(* IEC 61131-3 sources: github/ST定义, 5 files *)

(* ---- 座台定义.st ---- *)
TYPE E_NozzleState :
(
    (* 状态机枚举 *)
	eState_Idle,				// 空闲状态
	eState_Init,				// 初始化
	eState_NozzleIning,			// 座台进中(2段)
	eState_NozzleIned,			// 座台进完成
	eState_NozzleOuting,		// 座台退中(2段)
	eState_NozzleOuted,			// 座台退完成
	eState_Error				// 错误状态

);
END_TYPE

TYPE ST_NozzleSeg :
STRUCT

	(* 单段工艺参数 *)
	uiPres: UINT;		// 设定压力
	uiSpd: UINT;		// 设定速度
	udiPos: UDINT;		// 设定位置
	uiTime: UINT;		// 设定时间
	uiPresGrad: UINT;	// 设定压力斜率
	uiSpdGrad: UINT;	// 设定速度斜率

END_STRUCT
END_TYPE

TYPE ST_NozzlePara :
STRUCT

	(* 座台进工艺参数 21*)
	uiNozzleInSegCnt: UINT;							// 座台进段数选择
	uiNozzleInMode: UINT;							// 座台进方式选择 0:时间  1:行程  2:位置
	uiNozzleInLimitTime: UINT;						// 座台进限制时间
	aNozzleInSeg: ARRAY[1..2] OF ST_NozzleSeg;		// 座台进多段设定参数

	uiNozzleInPresStartGrad: UINT;				// 压力启动斜率
	uiNozzleInPresStopGrad: UINT;				// 压力停止斜率
	uiNozzleInSpdStartGrad: UINT;				// 速度启动斜率
	uiNozzleInSpdStopGrad: UINT;				// 速度停止斜率

	(* 座台退工艺参数 21*)
	uiNozzleOutSegCnt: UINT;							// 座台退段数选择
	uiNozzleOutMode: UINT;							// 座台退方式选择 0:时间  1:行程  2:位置
	uiNozzleOutLimitTime: UINT;						// 座台退限制时间
	aNozzleOutSeg: ARRAY[1..2] OF ST_NozzleSeg;		// 座台退多段设定参数

	uiNozzleOutPresStartGrad: UINT;				// 压力启动斜率
	uiNozzleOutPresStopGrad: UINT;				// 压力停止斜率
	uiNozzleOutSpdStartGrad: UINT;				// 速度启动斜率
	uiNozzleOutSpdStopGrad: UINT;				// 速度停止斜率

	(* 座台调试模式参数（调模状态下使用） *)
	stNozzleInDbgSeg: ST_NozzleSeg;				// 座台进调试段参数
	stNozzleOutDbgSeg: ST_NozzleSeg;			// 座台退调试段参数

END_STRUCT
END_TYPE

VAR_IN_OUT
	stNozzleAxis: ST_AxisRefHyd;
END_VAR
VAR_INPUT

    (* 控制命令 *)
	bStart: BOOL;				// 启动
	bStop: BOOL;				// 停止(有减速停)
	bEStop: BOOL;				// 急停(立即停止，无减速停)
	bReset: BOOL;				// 复位

    (* 模式选择 *)
	uiNozzleMode: UINT;		// 0:无模式 1:座台进模式 2:座台退模式 3:座台进(调试模式) 4:座台退(调试模式)

	(* 上位机设定参数输入 *)
	stNozzlePara: ST_NozzlePara;

	(* 数字信号输入 *)
	bNozzleInStop: BOOL;			// 座台进停止
	bNozzleOutStop: BOOL;			// 座台退停止

	(* 模拟信号输入 *)
	udiNozzleElecRulerVal: UDINT;			// 座台电子尺值

END_VAR
VAR_OUTPUT

	(* 状态输出 *)
	bBusy: BOOL;		// 忙状态
	bDone: BOOL;		// 完成状态
	bAlarm: BOOL;		// 报警状态

    (* 报警信息 *)
	dwAlarmID: DWORD;		// 报警代码（按位标识，可同时报告多个报警）
							(*	Bit0(1):   座台进超时
								Bit1(2):   座台退超时
								Bit2(4):   位置超限
								Bit3(8):   传感器异常
								...其他位预留
							*)

    (* 动作提示 *)
	uiActHint: UINT;		// 当前动作状态
							(*	0:无动作	1:报警状态	  2:座台进完成  3:座台退完成
								10: 		11:座台进1段  12:座台进2段	13:
								20:			21:座台退1段  22:座台退2段  23:
							*)
	uiActTime: UINT;		// 当前动作运行时间

	(* 动作状态输出 *)
	bNozzleIned: BOOL;		// 座台进完成
	bNozzleOuted: BOOL;		// 座台退完成

    (* 控制命令输出 *)
	uiPresCmd: UINT;		// 压力命令输出
	uiSpdCmd: UINT;			// 速度命令输出
	udiPosCmd: UDINT;		// 位置命令输出

END_VAR

(* ---- 储料定义.st ---- *)
TYPE E_MeterState :
(
    (* 状态机枚举 *)
	eState_Idle,				// 空闲状态
	eState_Init,				// 初始化
	eState_Metering,			// 储料中(8段)
	eState_Metered,				// 储料完成
	eState_Error				// 错误状态

);
END_TYPE

TYPE ST_MeterSeg :
STRUCT

	(* 单段工艺参数 *)
	uiSPres: UINT;		// 设定压力
	uiBackPres: UINT;	// 设定背压
	uiSpd: UINT;		// 设定速度
	udiPos: UDINT;		// 设定位置
	uiPresGrad: UINT;	// 设定压力斜率
	uiSpdGrad: UINT;	// 设定速度斜率

END_STRUCT
END_TYPE

TYPE ST_MeterPara :
STRUCT

	(* 储料工艺参数 71*)
	uiMeterSegCnt: UINT;						// 储料段数选择
	uiMeterMode: UINT;							// 储料退方式选择 0:电子尺  1:行程
	uiMeterLimitTime: UINT;						// 储料限制时间
	aMeterSeg: ARRAY[1..8] OF ST_MeterSeg;		// 储料多段设定参数

	uiMeterPresStartGrad: UINT;			// 压力启动斜率
	uiMeterPresStopGrad: UINT;			// 压力停止斜率
	uiMeterSpdStartGrad: UINT;			// 速度启动斜率
	uiMeterSpdStopGrad: UINT;			// 速度停止斜率

END_STRUCT
END_TYPE

FUNCTION_BLOCK FB_Meter
VAR_IN_OUT
	stMeterAxis: ST_AxisRefHyd;
END_VAR
VAR_INPUT

    (* 控制命令 *)
	bStart: BOOL;				// 启动
	bStop: BOOL;				// 停止(有减速停)
	bEStop: BOOL;				// 急停(立即停止，无减速停)
	bReset: BOOL;				// 复位

    (* 模式选择 *)
// 	uiMeterMode: UINT;		// 0:无模式 1: 2: 3:

	(* 上位机设定参数输入 *)
	stMeterPara: ST_MeterPara;

	(* 数字信号输入 *)
	bMeterStop: BOOL;			// 储料停止

	(* 模拟信号输入 *)
	udiInjElecRulerVal: UDINT;			// 射胶电子尺值

END_VAR
VAR_OUTPUT

	(* 状态输出 *)
	bBusy: BOOL;		// 忙状态
	bDone: BOOL;		// 完成状态
	bAlarm: BOOL;		// 报警状态
    (* 报警信息 *)
	dwAlarmID: DWORD;		// 报警代码（按位标识，可同时报告多个报警）
							(*	Bit0(1):   储料超时
								Bit1(2):   位置超限
								...其他位预留
							*)

    (* 动作提示 *)
	uiActHint: UINT;		// 当前动作状态
							(*	0:无动作  1:报警状态  2:储料完成    3:
								10: 	  11:储料1段  12:储料2段	13: 储料3段  14:储料4段    15:储料5段  16: 储料6段  17:储料7段   18:储料8段
							*)
	uiActTime: UINT;		// 当前动作运行时间

	(* 动作状态输出 *)
	bMetered: BOOL;				//储料完成

    (* 控制命令输出 *)
	uiPresCmd: UINT;		// 压力命令输出
	uiBackPresCmd: UINT;	// 背压命令输出
	uiSpdCmd: UINT;			// 速度命令输出
	udiPosCmd: UDINT;		// 位置命令输出

END_VAR

(* ---- 开合模定义.st ---- *)
(*
 * 文件: 开合模定义.st
 * 版本: V1.1
 *
 * 版本历史:
 * V1.0  2026-03-27  初始版本
 * V1.1  2026-04-02  新增调试模式支持(stOpenDebug/stCloseDebug)
 *
 * 说明: 开合模机构控制的功能块和数据结构定义
 *)

TYPE E_AxisState :
(
	Idle,				// 空闲状态
	Running,				// 运行状态
	Stop					// 停止状态
);
END_TYPE

TYPE E_ClampState :
(
	(* 状态机枚举 *)
	eState_Idle,				// 空闲状态
	eState_Init,				// 初始化
	eState_OpenUnload,			// 开模卸荷
	eState_Opening,				// 开模中(5段)
	eState_Opened,				// 开模完成
	eState_Closing,				// 合模中(3段)
	eState_Closed,				// 合模完成
	eState_CloseLowPress,		// 合模低压
	eState_CloseHighPress,		// 合模高压
	eState_Error				// 错误状态
);
END_TYPE

TYPE ST_PumpRequest :
STRUCT
	bRequest: BOOL;			// 泵请求
	rFlowSet: LREAL;		// 流量设定
	rPressureSet: LREAL;	// 压力设定
END_STRUCT
END_TYPE

TYPE ST_AxisRefHyd :
STRUCT
	(* 静态参数 *)
	bActive: BOOL;					// 轴是否激活
	eAxisState: E_AxisState;		// 轴状态
	nAxisID: INT;					// 轴ID号
	rMaxCylinderStroke: LREAL;		// 最大油缸行程
	rMaxVelocity: LREAL;			// 最大速度
	rMaxPressure: LREAL;			// 最大压力

	(* 运行设定值 *)
	rSetPosition: LREAL;				// 目标位置
	rSetVelocity: LREAL;			// 目标速度
	rSetPressure: LREAL;			// 目标压力

	(* 运行实际值 *)
	rActualPosition: LREAL;			// 实际位置
	rActualVelocity: LREAL;			// 实际速度
	rActualPressure: LREAL;			// 实际压力

	(* 泵请求 *)
	stPumpRequest: ST_PumpRequest;	// 向泵发送的请求

	(* 故障信息 *)
	nFaultCode: INT;					// 故障码
END_STRUCT
END_TYPE

TYPE ST_ClampSeg :
STRUCT

	(* 单段工艺参数 *)
	uiPres: UINT;		// 设定压力
	uiSpd: UINT;		// 设定速度
	udiPos: UDINT;		// 设定位置
	uiTime: UINT;		// 设定时间
	uiPresGrad: UINT;	// 设定压力斜率
	uiSpdGrad: UINT;	// 设定速度斜率

END_STRUCT
END_TYPE

TYPE ST_ClampPara :
STRUCT

	(* 开模工艺参数 *)
	uiOpenSegCnt: UINT;							// 开模段数选择 (1-5段)
	uiOpenMode: UINT;							// 开模方式选择 0:电子尺  1:行程
	uiOpenLimitTime: UINT;						// 开模限制时间
	stOpenUnloadPres: ST_ClampSeg;				// 开模卸荷设定参数
	aOpenSeg: ARRAY[1..5] OF ST_ClampSeg;		// 开模多段设定参数

	uiOpenPresStartGrad: UINT;					// 开模压力启动斜率
	uiOpenPresStopGrad: UINT;					// 开模压力停止斜率
	uiOpenSpdStartGrad: UINT;					// 开模速度启动斜率
	uiOpenSpdStopGrad: UINT;					// 开模速度停止斜率

	(* 合模工艺参数 *)
	uiCloseSegCnt: UINT;							// 合模段数选择 (1-3段)
	uiCloseMode: UINT;							// 合模方式选择 0:电子尺  1:行程
	uiCloseLimitTime: UINT;						// 合模限制时间
	uiCloseLowPresLimitTime: UINT;					// 合模低压保护时间
	uiCloseEndMode: UINT;							// 合模终止方式选择 0:时间 1:行程 2:压力
	uiCloseEndHighPres: UINT;						// 合模高压压力
	aCloseSeg: ARRAY[1..3] OF ST_ClampSeg;		// 合模多段设定参数
	stCloseLowPres: ST_ClampSeg;					// 合模低压设定参数
	stCloseHighPres: ST_ClampSeg;					// 合模高压设定参数

	uiClosePresStartGrad: UINT;					// 合模压力启动斜率
	uiClosePresStopGrad: UINT;					// 合模压力停止斜率
	uiCloseSpdStartGrad: UINT;					// 合模速度启动斜率
	uiCloseSpdStopGrad: UINT;					// 合模速度停止斜率

	(* 调试模式参数（调模状态下使用） *)
	stOpenDebug: ST_ClampSeg;					// 开模调试参数
	stCloseDebug: ST_ClampSeg;					// 合模调试参数

	(* 中子控制参数 *)
	aCoreFn: ARRAY[1..8] OF UINT;				// 中子功能 0:不使用 1:使用
	aCoreInMode: ARRAY[1..8] OF UINT;			// 中子进开始方式 0:行程 1:位置
	aCoreInStroke: ARRAY[1..8] OF UINT;		// 中子进开始行程
	aCoreInPos: ARRAY[1..8] OF UDINT;			// 中子进开始位置
	aCoreOutMode: ARRAY[1..8] OF UINT;			// 中子退开始方式 0:行程 1:位置
	aCoreOutStroke: ARRAY[1..8] OF UINT;		// 中子退开始行程
	aCoreOutPos: ARRAY[1..8] OF UDINT;			// 中子退开始位置

END_STRUCT
END_TYPE

FUNCTION_BLOCK FB_Clamp
VAR_IN_OUT
	ClampAxis: ST_AxisRefHyd;
END_VAR
VAR_INPUT

	(* 控制命令 *)
	bStart: BOOL;				// 启动
	bStop: BOOL;				// 停止(有减速停)
	bEStop: BOOL;				// 急停(立即停止，无减速停)
	bReset: BOOL;				// 复位

	(* 模式选择 *)
	uiClampMode: UINT;			// 0:无模式 1:开模模式 2:合模模式 3:开模(调试模式) 4:合模(调试模式)

	(* 上位机设定参数输入 *)
	stClampPara: ST_ClampPara;

	(* 数字信号输入 *)
	bOpenStop: BOOL;				// 开模停止
	bCloseLowPres: BOOL;			// 合模低压
	bCloseHighPres: BOOL;			// 合模高压
	bCloseStop: BOOL;				// 合模停止

	(* 模拟信号输入 *)
	udiClampElecRulerVal: UDINT;			// 锁模电子尺值
	uiClampPresElecRulerVal: UINT;			// 锁模压力值

END_VAR
VAR_OUTPUT

	(* 状态输出 *)
	bBusy: BOOL;		// 忙状态
	bDone: BOOL;		// 完成状态
	bAlarm: BOOL;		// 报警状态

	(* 报警信息 *)
	dwAlarmID: DWORD;		// 报警代码（按位标识，可同时报告多个报警）
							(*	Bit0(1):   低压保护超时
								Bit1(2):   开模超时
								Bit2(4):   合模超时
								Bit3(8):   位置超限
								Bit4(16):  传感器异常
								...其他位预留
							*)

	(* 动作提示 *)
	uiActHint: UINT;		// 当前动作状态
							(*	0:无动作	1:报警状态	2:开模完成  3:合模完成  4:中子执行
								10:开模卸荷	11:开模1段  12:开模2段	13:开模3段  14:开模4段  15:开模5段
								21:合模1段	22:合模2段  23:合模3段
								30:合模低压	31:合模高压
								40:开模调试	41:合模调试
							*)
	uiActTime: UINT;		// 当前动作运行时间
	bMoldOpened: BOOL;		// 开模完成
	bMoldClosed: BOOL;		// 合模完成
	aCoreAllow: ARRAY[1..8] OF BOOL;		// 中子允许信号（1..8组）

	(* 输出命令 *)
	uiPresCmd: UINT;		// 压力命令输出
	uiSpdCmd: UINT;		// 速度命令输出
	udiPosCmd: UDINT;		// 位置命令输出

END_VAR

(* ---- 液压伺服.st ---- *)
TYPE ST_AxisRefHyd :
STRUCT
	// ================================
	// AXIS_REF 轴索引结构体【完整版】
	// 包含：轴所有状态、位置、速度、扭矩、限位、报警、参数
	// ================================

    // ========== 1. 轴基础信息 ==========
    AxisNo           : INT;          // 轴编号 (0,1,2,3...)
    AxisName         : STRING[32];   // 轴名称
    Valid            : BOOL;         // 轴结构体有效
    AxisRefId        : UINT;         // 内部轴ID

    // ========== 2. 轴使能与状态 ==========
    Enabled          : BOOL;         // 轴已使能
    PowerOn          : BOOL;         // 伺服已上电
    Faulted          : BOOL;         // 轴故障
    Ready            : BOOL;         // 轴准备就绪
    Stopped          : BOOL;         // 轴已停止
    Moving           : BOOL;         // 轴正在运动
    Homing           : BOOL;         // 正在回零
    HomingDone       : BOOL;         // 回零完成
    InPosition       : BOOL;         // 已到达目标位置

    // ========== 3. 控制模式 ==========
    ControlMode      : INT;          // 当前控制模式
    // 0=未激活 1=位置 2=速度 3=扭矩 4=回零
    HomingMode       : INT;          // 回零模式

    // ========== 4. 位置数据 ==========
    ActualPosition   : LREAL;        // 实际位置（实时）
    CommandPosition  : LREAL;        // 指令位置
    HomePosition     : LREAL;        // 原点位置
    TargetPosition   : LREAL;        // 目标位置

    // ========== 5. 速度数据 ==========
    ActualVelocity   : LREAL;        // 实际速度
    CommandVelocity  : LREAL;        // 指令速度
    MaxVelocity      : LREAL;        // 轴最大速度

    // ========== 6. 加速度数据 ==========
    Acceleration     : LREAL;        // 当前加速度
    Deceleration     : LREAL;        // 当前减速度
    MaxAcceleration  : LREAL;        // 最大加速度
    MaxDeceleration  : LREAL;        // 最大减速度
    Jerk             : LREAL;        // 跃度
    MaxJerk          : LREAL;        // 最大跃度

    // ========== 7. 扭矩/力矩数据 ==========
    ActualTorque     : LREAL;        // 实际扭矩
    MaxTorque        : LREAL;        // 最大扭矩
    TorqueLimit      : LREAL;        // 扭矩限制

    // ========== 8. 限位信号 ==========
    PositiveLimit    : BOOL;         // 正限位触发
    NegativeLimit    : BOOL;         // 负限位触发
    SoftPlusLimit    : BOOL;         // 软正限位
    SoftNegLimit     : BOOL;         // 软负限位

    // ========== 9. 错误与报警 ==========
    Error            : BOOL;         // 轴错误
    ErrorId          : DWORD;        // 错误代码
    DriveAlarm       : BOOL;         // 驱动器报警
    DriveErrorId     : DWORD;        // 驱动器错误码
    ErrorStop        : BOOL;         // 错误停止

    // ========== 10. 状态字 ==========
    AxisStatus       : DWORD;        // 轴状态字
    DriveStatus      : DWORD;        // 驱动器状态字
    StatusBits       : ARRAY[0..15] OF BOOL; // 状态位

	(* 根据实际需求可以增加变量	*)

    // 1. 几何尺寸
    Bore_Dia        : LREAL;  // 缸径 mm
    Rod_Dia         : LREAL;  // 杆径 mm
    Stroke          : LREAL;  // 总行程 mm
    Min_Len         : LREAL;  // 最小安装距
    Max_Len         : LREAL;  // 最大安装距

    // 2. 面积容积
    Area_Piston     : LREAL;  // mm²
    Area_Rod        : LREAL;  // mm²
    Area_Annular    : LREAL;  // mm²
    Vol_Per_MM      : LREAL;  // mL/mm

    // 3. 压力推力
    Press_Rated     : LREAL;  // MPa
    Press_Max       : LREAL;  // MPa
    Force_Extend    : LREAL;  // N
    Force_Retract   : LREAL;  // N
    Effi            : LREAL;  // 效率

    // 4. 速度流量
    Vel_Ext_Max     : LREAL;  // mm/s
    Vel_Ret_Max     : LREAL;  // mm/s
    Flow_Ext        : LREAL;  // L/min
    Flow_Ret        : LREAL;  // L/min

    // 5. 位置限位
    Soft_Limit_F    : LREAL;  // 正向软限位
    Soft_Limit_B    : LREAL;  // 反向软限位
    Home_Pos        : LREAL;  // 原点位置
    Pos_Tolerance   : LREAL;  // 定位允差

    // 6. 负载摩擦
    Friction        : LREAL;
    Max_Axial_Load  : LREAL;
    Max_Rad_Load    : LREAL;

END_STRUCT
END_TYPE

FUNCTION_BLOCK FB_AxisHyd
VAR_IN_OUT
	stAxisHyd: ST_AxisRefHyd;
END_VAR
VAR_INPUT

    (* 控制命令 *)
	bStart: BOOL;		// 启动
	bStop: BOOL;		// 停止(有减速停)
	bEStop: BOOL;		// 急停(立即停止，无减速停)
	bReset: BOOL;		// 复位
	bDir: BOOL;			// 方向

    (* 模式选择 *)
	uiMode: UINT;		// 0:无模式 1:位置模式 2:速度模式 3:扭矩模式

    (* 参数设定 *)
	uiCmdPres  : UINT; 	// 压力目标
    uiSpd      : UINT; 	// 速度目标
    udiPos     : UDINT; // 位置目标
    uiForce    : UINT; 	// 力目标，可选(锁模,射胶时使用）

    uiAcc	: UINT;     // 加速度
    uiDec	: UINT;     // 减速度
	uiJerk	: UINT;     // 加加速

END_VAR
VAR_OUTPUT

	(* 状态输出 *)
	bBusy: BOOL;		// 忙状态
	bDone: BOOL;		// 完成状态
	bAlarm: BOOL;		// 报警状态

    (* 报警信息 *)
	dwAlarmID: DWORD;		// 报警代码
							(*	0:无
							*)

END_VAR
VAR
	// 状态机状态
	State: INT;
	// 内部状态
	StartOld: BOOL;
	StopOld: BOOL;
	EStopOld: BOOL;
	ResetOld: BOOL;
	// 位置/速度模拟
	SimPosition: LREAL;
	SimVelocity: LREAL;
	SimTorque: LREAL;
END_VAR

TYPE EN_AxisState =
(
	AXIS_IDLE		:= 0,	// 空闲
	AXIS_STARTING	:= 1,	// 启动中
	AXIS_RUNNING	:= 2,	// 运行中
	AXIS_STOPPING	:= 3,	// 停止中
	AXIS_STOPPED	:= 4,	// 已停止
	AXIS_ESTOPPING	:= 5,	// 急停中
	AXIS_ERROR		:= 6,	// 错误状态
	AXIS_RESETTING	:= 7	// 复位中
);
END_TYPE

(*
===================================================================
FB_AxisHyd - 液压伺服轴功能块【简化版】
===================================================================
功能：提供液压伺服轴的基本控制接口，用于PLC编程验证
备注：实际驱动器通信部分待后续实现

使用方式：
1. 配置 stAxisHyd 中的轴参数（行程、限位等）
2. 设置 uiMode 选择控制模式
3. 设置目标值（uiCmdPres, uiSpd, udiPos, uiForce）
4. 置位 bStart 启动轴运动
5. 监控 bBusy/bDone/bAlarm 状态

模式说明：
- uiMode=1: 位置模式 - 运动到 udiPos 指定位置
- uiMode=2: 速度模式 - 以 uiSpd 指定速度运动
- uiMode=3: 扭矩模式 - 以 uiForce 指定力运动
===================================================================
*)
FB_AxisHyd();

// 状态机
CASE State OF
	// ==================== 空闲状态 ====================
	AXIS_IDLE:
		bBusy		:= FALSE;
		bDone		:= FALSE;
		stAxisHyd.Moving	:= FALSE;
		stAxisHyd.Stopped	:= TRUE;

		// 检测启动命令
		IF bStart AND NOT StartOld THEN
			// 检查急停和报警
			IF stAxisHyd.DriveAlarm THEN
				dwAlarmID	:= 16#0001;	// 驱动器报警
				bAlarm		:= TRUE;
				State		:= AXIS_ERROR;
			ELSIF stAxisHyd.PositiveLimit AND bDir THEN
				dwAlarmID	:= 16#0002;	// 正限位
				bAlarm		:= TRUE;
				State		:= AXIS_ERROR;
			ELSIF stAxisHyd.NegativeLimit AND NOT bDir THEN
				dwAlarmID	:= 16#0003;	// 负限位
				bAlarm		:= TRUE;
				State		:= AXIS_ERROR;
			ELSE
				// 进入启动
				State		:= AXIS_STARTING;
			END_IF
		END_IF

	// ==================== 启动中 ====================
	AXIS_STARTING:
		bBusy		:= TRUE;
		stAxisHyd.Moving	:= TRUE;
		stAxisHyd.Stopped	:= FALSE;

		// 初始化模拟位置
		SimPosition	:= stAxisHyd.ActualPosition;
		SimVelocity	:= 0.0;
		SimTorque	:= 0.0;

		// 模式选择
		CASE uiMode OF
			1: // 位置模式
				stAxisHyd.TargetPosition	:= LREAL(udiPos) / 1000.0; // 单位转换
				stAxisHyd.CommandVelocity	:= LREAL(uiSpd) / 1000.0;
				stAxisHyd.CommandPosition	:= stAxisHyd.TargetPosition;

			2: // 速度模式
				SimVelocity	:= LREAL(uiSpd) / 1000.0;

			3: // 扭矩模式
				SimTorque	:= LREAL(uiForce) / 1000.0;

			ELSE
				dwAlarmID	:= 16#0010;	// 无效模式
				bAlarm		:= TRUE;
				State		:= AXIS_ERROR;
		END_CASE

		State	:= AXIS_RUNNING;

	// ==================== 运行中 ====================
	AXIS_RUNNING:
		bBusy		:= TRUE;
		stAxisHyd.Moving	:= TRUE;
		stAxisHyd.Stopped	:= FALSE;
		stAxisHyd.InPosition	:= FALSE;

		// 急停检测
		IF bEStop AND NOT EStopOld THEN
			State	:= AXIS_ESTOPPING;
		// 停止命令
		ELSIF bStop AND NOT StopOld THEN
			State	:= AXIS_STOPPING;
		// 位置模式到位检测
		ELSIF uiMode = 1 THEN
			SimPosition	:= SimPosition + SimVelocity * 0.05; // 模拟位置变化
			stAxisHyd.ActualPosition	:= SimPosition;

			// 到位判断
			IF ABS(SimPosition - stAxisHyd.TargetPosition) <= stAxisHyd.Pos_Tolerance THEN
				State	:= AXIS_STOPPED;
			END_IF
		// 速度/扭矩模式需要外部停止
		ELSE
			// 模拟运动
			IF bDir THEN
				SimPosition	:= SimPosition + SimVelocity * 0.05;
			ELSE
				SimPosition	:= SimPosition - SimVelocity * 0.05;
			END_IF
			stAxisHyd.ActualPosition	:= SimPosition;
		END_IF

	// ==================== 停止中 ====================
	AXIS_STOPPING:
		bBusy		:= TRUE;
		SimVelocity	:= SimVelocity * 0.8; // 减速

		IF ABS(SimVelocity) < 0.001 THEN
			SimVelocity	:= 0.0;
			stAxisHyd.ActualVelocity	:= 0.0;
			State	:= AXIS_STOPPED;
		ELSE
			SimPosition	:= SimPosition + SimVelocity * 0.05;
			stAxisHyd.ActualPosition	:= SimPosition;
			stAxisHyd.ActualVelocity	:= SimVelocity;
		END_IF

	// ==================== 已停止 ====================
	AXIS_STOPPED:
		bBusy		:= FALSE;
		bDone		:= TRUE;
		stAxisHyd.Moving	:= FALSE;
		stAxisHyd.Stopped	:= TRUE;
		stAxisHyd.InPosition	:= TRUE;
		SimVelocity	:= 0.0;
		SimTorque	:= 0.0;

		// 重新检测启动
		IF NOT bStart THEN
			State	:= AXIS_IDLE;
		END_IF

	// ==================== 急停中 ====================
	AXIS_ESTOPPING:
		bBusy		:= FALSE;
		bDone		:= FALSE;
		stAxisHyd.Moving	:= FALSE;
		SimVelocity	:= 0.0;
		SimTorque	:= 0.0;
		State	:= AXIS_STOPPED;

	// ==================== 错误状态 ====================
	AXIS_ERROR:
		bBusy		:= FALSE;
		bDone		:= FALSE;
		bAlarm		:= TRUE;
		stAxisHyd.Error	:= TRUE;
		stAxisHyd.ErrorId	:= dwAlarmID;
		stAxisHyd.Moving	:= FALSE;
		SimVelocity	:= 0.0;

		// 复位检测
		IF bReset AND NOT ResetOld THEN
			dwAlarmID	:= 0;
			bAlarm		:= FALSE;
			stAxisHyd.Error	:= FALSE;
			stAxisHyd.ErrorId	:= 0;
			State	:= AXIS_RESETTING;
		END_IF

	// ==================== 复位中 ====================
	AXIS_RESETTING:
		State	:= AXIS_IDLE;

END_CASE

// 边沿检测
StartOld	:= bStart;
StopOld		:= bStop;
EStopOld	:= bEStop;
ResetOld	:= bReset;

// 实时更新状态
stAxisHyd.ControlMode	:= INT_TO_UINT(uiMode);
stAxisHyd.Ready		:= (State = AXIS_IDLE) OR (State = AXIS_STOPPED);
stAxisHyd.Faulted	:= (State = AXIS_ERROR);

// 模拟实际值更新
stAxisHyd.CommandPosition	:= SimPosition;
stAxisHyd.CommandVelocity	:= SimVelocity;
stAxisHyd.ActualVelocity	:= SimVelocity;
stAxisHyd.ActualTorque		:= SimTorque;
stAxisHyd.PowerOn	:= TRUE;
stAxisHyd.Enabled	:= NOT bEStop;

END_FUNCTION_BLOCK

(* ---- 温度定义.st ---- *)
TYPE ST_EK312State :
(
	(* 状态机枚举 *)
	eState_Idle,				// 空闲状态
	eState_Init,				// 初始化
	eState_Heating,				// 加热中
	eState_Error				// 错误状态
);
END_TYPE

TYPE ST_EK312InSeg :
STRUCT

	(* 单段工艺参数 *)
	uiSetTemp: UINT;	// 温度设定值
	uiFunc: UINT;		// 温度设定功能 0:不用 1:使用
	uiP: UINT;			// 温度设定P值
	uiD: UINT;			// 温度设定D值
	uiMax: UINT;		// 温度设定上限
	uiMin: UINT;		// 温度设定下限

END_STRUCT
END_TYPE

TYPE ST_EK312InPara :
STRUCT

	(* EK312输入参数 123*)
	aSeg: ARRAY[1..12] OF ST_EK312InSeg;	// 多段输入参数
	aInputAddr: ARRAY[1..50] OF UINT;		//输入地址

    (* 配置参数 *)
	uiStationNo: UINT;			// 站号
	uiColorSelect: UINT;		// 单双三色选择  80
	uiAColor: UINT;				// A色开选择    81
	uiBColor: UINT;				// B色开选择    82
	uiCColor: UINT;				// C色开选择    83
	uiANozMode: UINT;			// A色射咀方式    17
	uiBNozMode: UINT;			// B色射咀方式    84
	uiCNozMode: UINT;			// C色射咀方式 	  86
	uiANozPerc: UINT;			// A色射咀百分比  22
	uiBNozPerc: UINT;			// B色射咀百分比  85
	uiCNozPerc: UINT;			// C色射咀百分比  87
	uiContSSR: UINT;			// 接触器和固态继电器选择    24
	uiNozCtrlCycle: UINT;		// 射咀控制周期    26

END_STRUCT
END_TYPE

TYPE ST_EK312OutSeg :
STRUCT

	(* 单段工艺参数 *)
	uiActualTemp: UINT;		// 温度实际值
	uiState: UINT;			// 温度状态值 0:正常 1:偏低 2:偏高 3:断线

END_STRUCT
END_TYPE

TYPE ST_EK312OutPara :
STRUCT

	(* EK312输出参数 124*)
	aSeg: ARRAY[1..12] OF ST_EK312OutSeg;		// 多段输出参数
	aOutputAddr: ARRAY[1..100] OF UINT;			//输出地址

END_STRUCT
END_TYPE

FUNCTION_BLOCK FB_EK312
VAR_INPUT

	(* 控制命令 *)
	bStart: BOOL;	// 启动
	bStop: BOOL;	// 停止
	bReset: BOOL;	// 复位

	(* 输出控制命令 *)
	bR0:BOOL;		// R0使能
	bR1:BOOL;		// R1使能
	bR2:BOOL;		// R2使能
	bR3:BOOL;		// R3使能

    (* 模式选择 *)
// 	uiMode: UINT;		// 0:无模式 1: 2: 3:

	(* EK312输入参数 *)
	stInPara: ST_EK312InPara;

END_VAR
VAR_OUTPUT

	(* 状态输出 *)
	bBusy: BOOL;		// 忙状态
	bDone: BOOL;		// 完成状态
	bAlarm: BOOL;		// 报警状态

    (* 报警信息 *)
	dwAlarmID: DWORD;		// 报警代码
							(*	0:无
								1000: 通讯失败
							*)

	(* EK312输出参数 *)
	stOutPara: ST_EK312OutPara;

    (* 加热状态输出 *)
	uiHeatState: UINT;		// 温度加热状态  220

	(* 版本号 *)
	uiVersion: UINT;		// 版本号  222

END_VAR
VAR
END_VAR
